{attribute 'qualified_only'}
VAR_GLOBAL
	
	// Systemzustand
	SysState			:INT;		// 0 = Grundfunktion nicht aktive | 1 = Grundfunktion aktive
	SekReady			:BOOL;		// Gibt an ob Sekundärreaktor bereit ist
	SekActiv			:BOOL;		// Gibt an ob Sekundärreaktor aktiv ist

	// Bedienparameter
	Bedien_Power		:BOOL;
	Bedien_Reset		:BOOL;
	
	// Debug-Variablen: 
	Debug_Verbunden		:BOOL := TRUE;
	Debug_Start			:BOOL := TRUE;
	Debug_SekStart		:BOOL;

END_VAR

(* stored: Version 1.1.0.1, ProductVersion 3.1.4024.12
   GVL GVL: Id {2f1a5837-5f08-48be-bb75-10432a2fbf59} *)
